// TIA Portal V19 export
DATA_BLOCK "MixingIngredientsCake"   // DB224
// stored: MemoryReserve 100
   VAR
      mixingCake { S7_SetPoint := 'True'} : "typeMixingIngredientsCake";
   END_VAR
BEGIN
END_DATA_BLOCK
